(* IEC 61131-3 sources: ST-sUtils/, 4 files *)

(* ---- U_sByte.st ---- *)
//Boris Spiridonov
//14.02.22
TYPE U_sByte:
UNION
  bytes:  ARRAY[0..0] OF BYTE;
  bits:   ARRAY[0..7] OF BOOL;
END_UNION
END_TYPE

(* ---- F_s_byte_to_bools.st ---- *)
//F_s_byte_to_bools
//Boris Spiridonov
//14.02.22
FUNCTION F_s_byte_to_bools : BOOL
VAR_EXTERNAL
END_VAR
VAR_INPUT
  In : BYTE;
END_VAR
VAR
  bools_tmp :  U_sByte;
  index :      INT;
END_VAR
VAR_OUTPUT
  Out :  ARRAY[0..7] OF BOOL;
END_VAR

  bools_tmp.bytes[0] := In;

  index := 0;

  FOR index := INT#0 TO INT#7 BY INT#1 DO
     Out[index] := bools_tmp.bits[index];
  END_FOR;
END_FUNCTION

(* ---- F_s_is_eip_error.st ---- *)
//F_s_is_eip_error
//Boris Spiridonov
//14.02.22
FUNCTION F_s_is_eip_error : BOOL
VAR_EXTERNAL
  _EIP1_TDLinkErr	: BOOL;
END_VAR
VAR_IN_OUT
  is_eip_error :    BOOL;
END_VAR

//TODO refactor add platform switcher
//Sysmac
  is_eip_error := _EIP1_TDLinkErr;

  F_is_eip_error := is_eip_error;
END_FUNCTION

(* ---- F_s_is_string_empty.st ---- *)
//F_s_is_string_empty
//Boris Spiridonov
//17.11.21
FUNCTION F_s_is_string_empty : BOOL
VAR_INPUT
  In : BYTE;
END_VAR
VAR
  string_tmp :	STRING[256];
  string_lenght :	UINT;
END_VAR
VAR_OUTPUT
  Out :      BOOL;
END_VAR

  string_tmp := TrimL(In);
  string_tmp := TrimR(string_tmp);

//TODO refactor add platform switcher
//Sysmac
  string_lenght := GetByteLen(string_tmp);

  Out := string_lenght < 1 ;
  F_s_is_string_empty := Out;
END_FUNCTION
